(* PLC project To_FTP_server, Beckhoff Automation GmbH TwinCAT PLC Control 3.5.13.20 *)
(* stored: creationDateTime 2020-09-10T09:40:10.3057489, modificationDateTime 2020-09-10T09:40:10.3057489 *)

FUNCTION_BLOCK FB_CreateMessage
VAR_INPUT
	stLoad		:ST_LoadData;
	bCreateMessage :BOOL;
END_VAR
VAR_OUTPUT
	sMessageOut:T_MaxString;
	bMessageReady:BOOL:=FALSE;
END_VAR
VAR
sTemplateMessage:T_MaxString:='|MsgNam=WMS.TEGEW|TrxId=|RFIDNAM=|DzTrn=|ArtGewBru=|';
fbPulsCreateMessage:R_TRIG;
sTrxId:STRING;
i :INT;
sMessage :T_MaxString;
iPosRFID:INT;
iPosTime:INT;
iPosBrutto:INT;
	fbTime : FB_LocalSystemTime;
	System_Time: DT;
	bEnableTime: BOOL := TRUE;
tNow : TIME;
sSystemTime:STRING;
sSystemTimeYear:STRING;
sSystemTimeMonth:STRING;

fbFileOpen:FB_FileOpen;
END_VAR
VAR PERSISTENT
iCountTrxId: UINT;
END_VAR

            fbTime  (bEnable :=bEnableTime , dwCycle :=1);
bEnableTime := FALSE;

System_Time := SYSTEMTIME_TO_DT (fbTime.systemTime);
sSystemTime := DT_TO_STRING (System_Time);
sSystemTime := MID (sSystemTime, 19, 4);
sSystemTimeYear :=LEFT(sSystemTime,4);
sSystemTimeMonth:=MID(sSystemTime,2,6);
sSystemTime := MID (sSystemTime, 11, 9);
sSystemTime:= REPLACE(sSystemTime,CONCAT('.',sSystemTimeMonth),1,3);
sSystemTime:= INSERT(sSystemTime,CONCAT(CONCAT('.',sSystemTimeYear),' '),5);




fbPulsCreateMessage(CLK:=bCreateMessage);

IF fbPulsCreateMessage.Q THEN
	iCountTrxId:= iCountTrxId+1;
	i:=1;
END_IF
CASE i OF
	0:  ;
	
	1:
bMessageReady:=FALSE;	
sTrxId:= INT_TO_STRING(iCountTrxId);	

sMessage:= INSERT(sTemplateMessage,	sTrxId,24);
iPosRFID:= FIND(sMessage,'RFIDNAM=');
sMessage:= INSERT(sMessage,	stLoad.sID,iPosRFID+7);
iPosTime:= FIND(sMessage,'DzTrn=');
sMessage:= INSERT(sMessage,	sSystemTime,iPosTime+5);
iPosBrutto:= FIND(sMessage,'ArtGewBru=');
sMessage:= INSERT(sMessage,	stLoad.sWeight,iPosBrutto+9);

	i:=3;
	
	3:
sMessageOut:=	sMessage;
IF 	sMessageOut=sMessage THEN
	bMessageReady:=TRUE;
	i:=0;
END_IF

	
END_CASE
          
END_FUNCTION_BLOCK
